// TIA Portal V19 export
FUNCTION_BLOCK "ISDU_Event Index 37"   // FB37, STL
TITLE = Read events over ISDU and split information
{ S7_Optimized_Access := 'TRUE' }
// stored: AutoNumber false, MemoryReserve 100
   VAR_INPUT
      IHW_hwID : HW_ANY;   // Start adress IO-Link master
      II_CAP : Int;   // Access-point IO-Link-Call funktion (see manual of the master e.g. Siemens 227)
      II_PORT : Int;   // Number of uses IO-Link-Port (see manual of the master)
   END_VAR
   VAR_IN_OUT
      IO_ReadReq : Bool;   // Request reading parameters (set by application / reset by FB)
   END_VAR
   VAR
      ReadAsyc : "LIOLink_Device";
      SST_RecordData : Array[0..231] of Byte;   // data area for reading / writing data (max. 232 byte)
   END_VAR
   VAR_TEMP
      FlagWork : Struct
         TEMP0_0 : Byte;
         TEMP0_1 : Byte;
         TEMP0_2 : Byte;
         TEMP0_3 : Byte;
      END_STRUCT;
      tmp_RET_VAL : Int;
   END_VAR
BEGIN

NETWORK
TITLE = Request reading parameters (set by application / reset by FB)
      CALL  #ReadAsyc
      ( execute       := #IO_ReadReq,
        hwID          := #IHW_hwID,
        cap           := #II_CAP,
        readWrite     := false,
        port          := #II_PORT,
        index         := 37,
        subindex      := 0,
        writeLen      := #ReadAsyc.writeLen,
        timeout       := #ReadAsyc.timeout,
        pollingPeriod := T#100ms,
        done          := #ReadAsyc.done,
        busy          := #ReadAsyc.busy,
        error         := #ReadAsyc.error,
        status        := #ReadAsyc.status,
        diagnostics   := #ReadAsyc.diagnostics,
        readLen       := #ReadAsyc.readLen,
        record        := #SST_RecordData
      );


      SET;
      R     #IO_ReadReq;




END_FUNCTION_BLOCK
